{attribute 'GeneratedUsingTerminal: EL9070--0000'}
{attribute addProperty BoxType "EL9070--0000"}
{attribute addProperty Description "EL9070 Shield terminal"}
{attribute addProperty Physics "KK"}
{attribute addProperty Id "EL9070"}
{attribute addProperty CRC "927637283"}
{attribute addProperty Size "0"}
TYPE EL9070_374A9F23 EXTENDS EtcSlaveTerminalBase_947E5A46 :
STRUCT
END_STRUCT
END_TYPE

(* stored: Version 1.2.0.0, ProductVersion 3.1.4024.11
   DUT EL9070_374A9F23: Id {faaecf2c-07da-4d53-ae3f-4e18c51d02aa} *)
